# EPICS autosave request: ADPcoWin/iocs/pcowinIOC/iocBoot/iocPcoWin/auto_settings.req
file "pco_settings.req", 		P=$(P), R=cam1:
file "NDStdArrays_settings.req",	P=$(P),	R=image1:
file "commonPlugin_settings.req",	P=$(P)
